FUNCTION_BLOCK PML_UdefinedState
VAR_INPUT
END_VAR
VAR_OUTPUT
END_VAR
VAR
END_VAR

END_FUNCTION_BLOCK

(* stored: Version 1.1.0.1, ProductVersion 3.1.4024.11
   POU PML_UdefinedState: Id {01122847-2515-4c38-9336-f3153f26aa0b}, SpecialFunc None *)
